PROGRAM main
  VAR
    Start_PB : BOOL;
    Stop_PB : BOOL;
    Machine : BOOL;
    Fan : BOOL;
    TOF0 : TOF;
  END_VAR

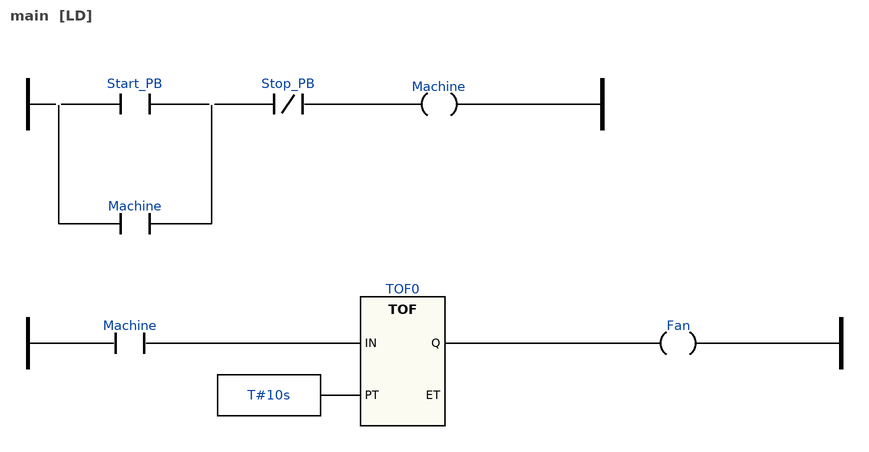
(* LD diagram, written out as Structured Text *)
Machine := (Machine OR Start_PB) AND NOT Stop_PB;
TOF0(IN := Machine, PT := T#10s);
Fan := TOF0.Q;
END_PROGRAM
